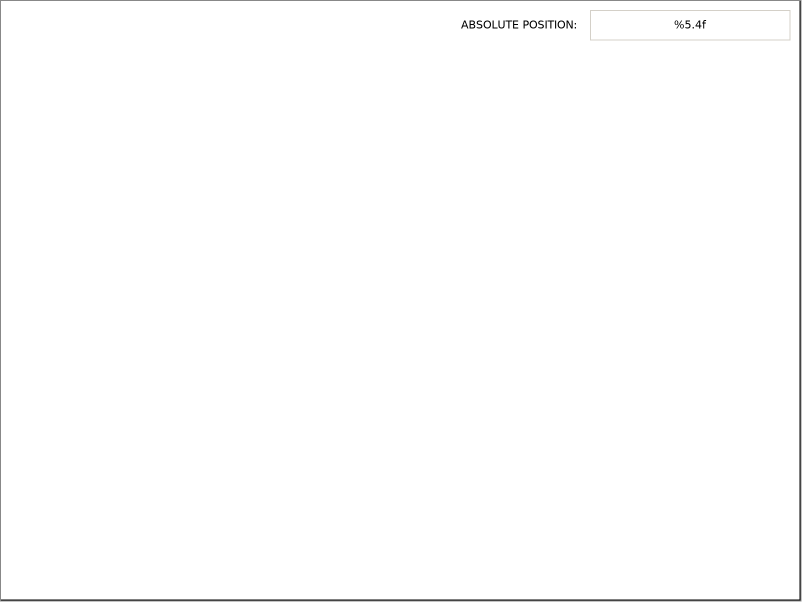
VISUALIZATION F28_Move_Absolute  // 802x602
    Rectangle (0,0 800x600)
    Textfield (590,10 200x30), "%5.4f", text variable: MAIN.axes[MAIN.hmiAxisSelect].POSITION
        OnMouseClick: write MAIN.axes[MAIN.hmiAxisSelect].POSITION via Default
    Label (410,10 170x30), "ABSOLUTE POSITION:"
END_VISUALIZATION

(* stored: Version 1.1.0.1, ProductVersion 3.1.4022.7
   Visu F28_Move_Absolute: Id {897b5cfa-5b97-48f9-8d85-37fa04ba33f6} *)
